// TwinCAT 3 PLC project Gamora
// ProgramVersion: 3.1.4026.1+972e9c44872ad038b353624a861fd7e3244e9f75
// libraries:
//   Tc2_Standard, * (Beckhoff Automation GmbH)
//   Tc2_System, * (Beckhoff Automation GmbH)
//   Tc2_Utilities, * (Beckhoff Automation GmbH)
// project tree:
//   / PlcTask.TcTTO (not stored)
//   POUs/EventLoggerExample/ FB_EventLogger.TcPOU
//   POUs/ MAIN.TcPOU

// ---- POUs/EventLoggerExample/FB_EventLogger.TcPOU
FUNCTION_BLOCK FB_EventLogger
VAR
	bBoolean : BOOL := FALSE;
	
	// Event example
	eEventType1 : E_EventType := E_EventType.Alarm;
	eEventSeverity1 : TcEventSeverity.Error;
	nEventIdentity1 : UDINT := 1;
	sEventText1 : STRING(255) := "This is an example";
	
	fbCsvPersistantEventStorage : FB_CsvPersistantEventStorage;
	fbEventLogger : FB_EventLogger(fbCsvPersistantEventStorage);
END_VAR

//Example of event
IF bBoolean THEN
	EventLogger.AddEvent(eEventType1, eEventSeverity1, nEventIdentity1, sEventText1);
END_IF

fbCsvPersistantEventStorage();

END_FUNCTION_BLOCK

// ---- POUs/MAIN.TcPOU
PROGRAM MAIN
VAR
	
END_VAR

END_PROGRAM
